FUNCTION_BLOCK FB_MovingHeadOffCommand IMPLEMENTS I_Command
VAR
	refMovingHead : REFERENCE TO FB_MovingHead;
END_VAR

METHOD Execute
IF (__ISVALIDREF(THIS^.refMovingHead)) THEN
	THIS^.refMovingHead.Off();
END_IF
END_METHOD

METHOD FB_init : BOOL
VAR_INPUT
	bInitRetains 	: BOOL; // if TRUE, the retain variables are initialized (warm start / cold start)
	bInCopyCode 	: BOOL;  // if TRUE, the instance afterwards gets moved into the copy code (online change)
	refMovingHead 	: REFERENCE TO FB_MovingHead;
END_VAR
IF (__ISVALIDREF(refMovingHead)) THEN
	THIS^.refMovingHead REF= refMovingHead;
ELSE
	THIS^.refMovingHead REF= 0;
END_IF
END_METHOD

END_FUNCTION_BLOCK

(* stored: Version 1.1.0.1, ProductVersion 3.1.4022.18
   POU FB_MovingHeadOffCommand: Id {7ac6b268-1904-407f-a3b1-73e26c02133d}, SpecialFunc None
   Method Execute: Id {ce92b5c6-96f3-4e1d-af6e-e2ef961a1197}
   Method FB_init: Id {749ea78c-4f44-4848-bdd0-2719517e87ce} *)
